{attribute addProperty BoxType ""}
{attribute addProperty Id "_defaultSyncUnitTasks_486549DC19524.3750"}
{attribute addProperty CRC "3400674619"}
{attribute addProperty SizeInBites "195"}
{attribute addProperty SizeInBytes "24.375"}
TYPE SyncUnits_CAB22D3B :
STRUCT
	{attribute addProperty Name "_default"}
	_default : SyncUnitTasks_486549DC;
END_STRUCT
END_TYPE

(* stored: Version 1.2.0.0, ProductVersion 3.1.4024.9
   DUT SyncUnits_CAB22D3B: Id {9fe97d18-5391-4292-800e-3a8efe86242c} *)
